Fanuc KAREL source: ka00053.KL

PROGRAM KA00053
%NOLOCKGROUP
VAR
SRC : POSITION;DST : POSITION
BEGIN
--
DST=SRC
END KA00053
